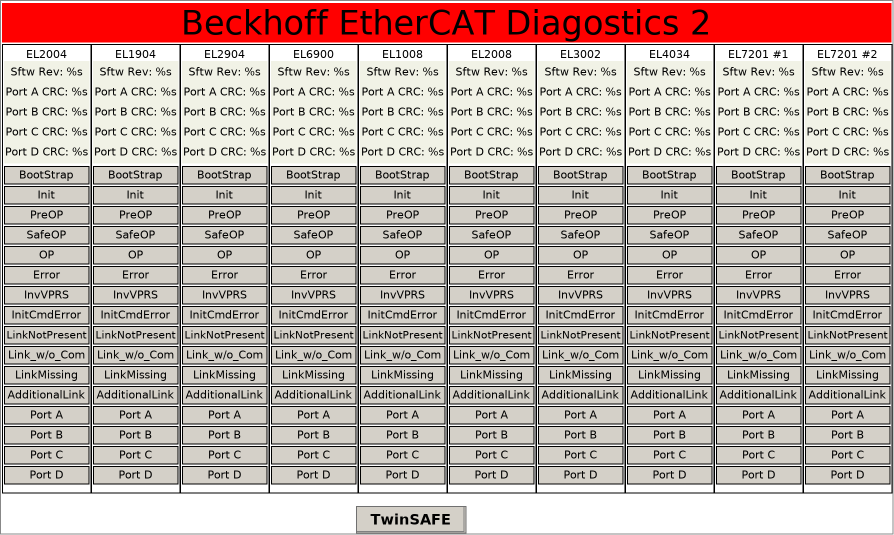
VISUALIZATION EtherCAT_Diag2  // 894x535
    Button (356,506 110x27), "TwinSAFE"
        OnMouseClick: change screen: TwinSAFE
    RoundedRectangle (2,3 889x39), "Beckhoff EtherCAT Diagostics 2"
    Group (2,42 89x451)
        RoundedRectangle (0,2 89x449)
        Label (2,0 85x25), "EL2004"
        Rectangle (2,19 85x22), "Sftw Rev: %s", text variable: g_iHMI_ProdCodeEL2004
        Rectangle (2,39 85x22), "Port A CRC: %s", text variable: g_stHMI_EL2004CrcErrorEx.portA
        Rectangle (2,59 85x22), "Port B CRC: %s", text variable: g_stHMI_EL2004CrcErrorEx.portB
        Rectangle (2,79 85x22), "Port C CRC: %s", text variable: g_stHMI_EL2004CrcErrorEx.portC
        Rectangle (2,99 85x22), "Port D CRC: %s", text variable: g_stHMI_EL2004CrcErrorEx.portD
        Rectangle (2,124 85x18), "BootStrap", colour toggle: g_stHMI_EL2004EcSlaveStateBits.bBootStrap
        Rectangle (2,144 85x18), "Init", colour toggle: g_stHMI_EL2004EcSlaveStateBits.bInit
        Rectangle (2,164 85x18), "PreOP", colour toggle: g_stHMI_EL2004EcSlaveStateBits.bPreop
        Rectangle (2,184 85x18), "SafeOP", colour toggle: g_stHMI_EL2004EcSlaveStateBits.bSafeOp
        Rectangle (2,204 85x18), "OP", colour toggle: g_stHMI_EL2004EcSlaveStateBits.bOp
        Rectangle (2,224 85x18), "Error", colour toggle: g_stHMI_EL2004EcSlaveStateBits.bError
        Rectangle (2,244 85x18), "InvVPRS", colour toggle: g_stHMI_EL2004EcSlaveStateBits.bInvVPRS
        Rectangle (2,264 85x18), "InitCmdError", colour toggle: g_stHMI_EL2004EcSlaveStateBits.bInitCmdError
        Rectangle (2,284 85x18), "LinkNotPresent", colour toggle: g_stHMI_EL2004EcSlaveStateBits.bLinkNotPresent
        Rectangle (2,304 85x18), "Link_w/o_Com", colour toggle: g_stHMI_EL2004EcSlaveStateBits.bLinkWithoutComm
        Rectangle (2,324 85x18), "LinkMissing", colour toggle: g_stHMI_EL2004EcSlaveStateBits.bLinkMissing
        Rectangle (2,344 85x18), "AdditionalLink", colour toggle: g_stHMI_EL2004EcSlaveStateBits.bAdditionalLink
        Rectangle (2,364 85x18), "Port A", colour toggle: g_stHMI_EL2004EcSlaveStateBits.bPortA
        Rectangle (2,384 85x18), "Port B", colour toggle: g_stHMI_EL2004EcSlaveStateBits.bPortB
        Rectangle (2,404 85x18), "Port C", colour toggle: g_stHMI_EL2004EcSlaveStateBits.bPortC
        Rectangle (2,424 85x18), "Port D", colour toggle: g_stHMI_EL2004EcSlaveStateBits.bPortD
    Group (91,42 89x451)
        RoundedRectangle (0,2 89x449)
        Label (2,0 85x25), "EL1904"
        Rectangle (2,19 85x22), "Sftw Rev: %s", text variable: g_iHMI_ProdCodeEL1904
        Rectangle (2,39 85x22), "Port A CRC: %s", text variable: g_stHMI_EL1904CrcErrorEx.portA
        Rectangle (2,59 85x22), "Port B CRC: %s", text variable: g_stHMI_EL1904CrcErrorEx.portB
        Rectangle (2,79 85x22), "Port C CRC: %s", text variable: g_stHMI_EL1904CrcErrorEx.portC
        Rectangle (2,99 85x22), "Port D CRC: %s", text variable: g_stHMI_EL1904CrcErrorEx.portD
        Rectangle (2,124 85x18), "BootStrap", colour toggle: g_stHMI_EL1904EcSlaveStateBits.bBootStrap
        Rectangle (2,144 85x18), "Init", colour toggle: g_stHMI_EL1904EcSlaveStateBits.bInit
        Rectangle (2,164 85x18), "PreOP", colour toggle: g_stHMI_EL1904EcSlaveStateBits.bPreop
        Rectangle (2,184 85x18), "SafeOP", colour toggle: g_stHMI_EL1904EcSlaveStateBits.bSafeOp
        Rectangle (2,204 85x18), "OP", colour toggle: g_stHMI_EL1904EcSlaveStateBits.bOp
        Rectangle (2,224 85x18), "Error", colour toggle: g_stHMI_EL1904EcSlaveStateBits.bError
        Rectangle (2,244 85x18), "InvVPRS", colour toggle: g_stHMI_EL1904EcSlaveStateBits.bInvVPRS
        Rectangle (2,264 85x18), "InitCmdError", colour toggle: g_stHMI_EL1904EcSlaveStateBits.bInitCmdError
        Rectangle (2,284 85x18), "LinkNotPresent", colour toggle: g_stHMI_EL1904EcSlaveStateBits.bLinkNotPresent
        Rectangle (2,304 85x18), "Link_w/o_Com", colour toggle: g_stHMI_EL1904EcSlaveStateBits.bLinkWithoutComm
        Rectangle (2,324 85x18), "LinkMissing", colour toggle: g_stHMI_EL1904EcSlaveStateBits.bLinkMissing
        Rectangle (2,344 85x18), "AdditionalLink", colour toggle: g_stHMI_EL1904EcSlaveStateBits.bAdditionalLink
        Rectangle (2,364 85x18), "Port A", colour toggle: g_stHMI_EL1904EcSlaveStateBits.bPortA
        Rectangle (2,384 85x18), "Port B", colour toggle: g_stHMI_EL1904EcSlaveStateBits.bPortB
        Rectangle (2,404 85x18), "Port C", colour toggle: g_stHMI_EL1904EcSlaveStateBits.bPortC
        Rectangle (2,424 85x18), "Port D", colour toggle: g_stHMI_EL1904EcSlaveStateBits.bPortD
    Group (180,42 89x451)
        RoundedRectangle (0,2 89x449)
        Label (2,0 85x25), "EL2904"
        Rectangle (2,19 85x22), "Sftw Rev: %s", text variable: g_iHMI_ProdCodeEL2904
        Rectangle (2,39 85x22), "Port A CRC: %s", text variable: g_stHMI_EL2904CrcErrorEx.portA
        Rectangle (2,59 85x22), "Port B CRC: %s", text variable: g_stHMI_EL2904CrcErrorEx.portB
        Rectangle (2,79 85x22), "Port C CRC: %s", text variable: g_stHMI_EL2904CrcErrorEx.portC
        Rectangle (2,99 85x22), "Port D CRC: %s", text variable: g_stHMI_EL2904CrcErrorEx.portD
        Rectangle (2,124 85x18), "BootStrap", colour toggle: g_stHMI_EL2904EcSlaveStateBits.bBootStrap
        Rectangle (2,144 85x18), "Init", colour toggle: g_stHMI_EL2904EcSlaveStateBits.bInit
        Rectangle (2,164 85x18), "PreOP", colour toggle: g_stHMI_EL2904EcSlaveStateBits.bPreop
        Rectangle (2,184 85x18), "SafeOP", colour toggle: g_stHMI_EL2904EcSlaveStateBits.bSafeOp
        Rectangle (2,204 85x18), "OP", colour toggle: g_stHMI_EL2904EcSlaveStateBits.bOp
        Rectangle (2,224 85x18), "Error", colour toggle: g_stHMI_EL2904EcSlaveStateBits.bError
        Rectangle (2,244 85x18), "InvVPRS", colour toggle: g_stHMI_EL2904EcSlaveStateBits.bInvVPRS
        Rectangle (2,264 85x18), "InitCmdError", colour toggle: g_stHMI_EL2904EcSlaveStateBits.bInitCmdError
        Rectangle (2,284 85x18), "LinkNotPresent", colour toggle: g_stHMI_EL2904EcSlaveStateBits.bLinkNotPresent
        Rectangle (2,304 85x18), "Link_w/o_Com", colour toggle: g_stHMI_EL2904EcSlaveStateBits.bLinkWithoutComm
        Rectangle (2,324 85x18), "LinkMissing", colour toggle: g_stHMI_EL2904EcSlaveStateBits.bLinkMissing
        Rectangle (2,344 85x18), "AdditionalLink", colour toggle: g_stHMI_EL2904EcSlaveStateBits.bAdditionalLink
        Rectangle (2,364 85x18), "Port A", colour toggle: g_stHMI_EL2904EcSlaveStateBits.bPortA
        Rectangle (2,384 85x18), "Port B", colour toggle: g_stHMI_EL2904EcSlaveStateBits.bPortB
        Rectangle (2,404 85x18), "Port C", colour toggle: g_stHMI_EL2904EcSlaveStateBits.bPortC
        Rectangle (2,424 85x18), "Port D", colour toggle: g_stHMI_EL2904EcSlaveStateBits.bPortD
    Group (269,42 89x451)
        RoundedRectangle (0,2 89x449)
        Label (2,0 85x25), "EL6900"
        Rectangle (2,19 85x22), "Sftw Rev: %s", text variable: g_iHMI_ProdCodeEL6900
        Rectangle (2,39 85x22), "Port A CRC: %s", text variable: g_stHMI_EL6900CrcErrorEx.portA
        Rectangle (2,59 85x22), "Port B CRC: %s", text variable: g_stHMI_EL6900CrcErrorEx.portB
        Rectangle (2,79 85x22), "Port C CRC: %s", text variable: g_stHMI_EL6900CrcErrorEx.portC
        Rectangle (2,99 85x22), "Port D CRC: %s", text variable: g_stHMI_EL6900CrcErrorEx.portD
        Rectangle (2,124 85x18), "BootStrap", colour toggle: g_stHMI_EL6900EcSlaveStateBits.bBootStrap
        Rectangle (2,144 85x18), "Init", colour toggle: g_stHMI_EL6900EcSlaveStateBits.bInit
        Rectangle (2,164 85x18), "PreOP", colour toggle: g_stHMI_EL6900EcSlaveStateBits.bPreop
        Rectangle (2,184 85x18), "SafeOP", colour toggle: g_stHMI_EL6900EcSlaveStateBits.bSafeOp
        Rectangle (2,204 85x18), "OP", colour toggle: g_stHMI_EL6900EcSlaveStateBits.bOp
        Rectangle (2,224 85x18), "Error", colour toggle: g_stHMI_EL6900EcSlaveStateBits.bError
        Rectangle (2,244 85x18), "InvVPRS", colour toggle: g_stHMI_EL6900EcSlaveStateBits.bInvVPRS
        Rectangle (2,264 85x18), "InitCmdError", colour toggle: g_stHMI_EL6900EcSlaveStateBits.bInitCmdError
        Rectangle (2,284 85x18), "LinkNotPresent", colour toggle: g_stHMI_EL6900EcSlaveStateBits.bLinkNotPresent
        Rectangle (2,304 85x18), "Link_w/o_Com", colour toggle: g_stHMI_EL6900EcSlaveStateBits.bLinkWithoutComm
        Rectangle (2,324 85x18), "LinkMissing", colour toggle: g_stHMI_EL6900EcSlaveStateBits.bLinkMissing
        Rectangle (2,344 85x18), "AdditionalLink", colour toggle: g_stHMI_EL6900EcSlaveStateBits.bAdditionalLink
        Rectangle (2,364 85x18), "Port A", colour toggle: g_stHMI_EL6900EcSlaveStateBits.bPortA
        Rectangle (2,384 85x18), "Port B", colour toggle: g_stHMI_EL6900EcSlaveStateBits.bPortB
        Rectangle (2,404 85x18), "Port C", colour toggle: g_stHMI_EL6900EcSlaveStateBits.bPortC
        Rectangle (2,424 85x18), "Port D", colour toggle: g_stHMI_EL6900EcSlaveStateBits.bPortD
    Group (358,42 89x451)
        RoundedRectangle (0,2 89x449)
        Label (2,0 85x25), "EL1008"
        Rectangle (2,19 85x22), "Sftw Rev: %s", text variable: g_iHMI_ProdCodeEL1008
        Rectangle (2,39 85x22), "Port A CRC: %s", text variable: g_stHMI_EL1008CrcErrorEx.portA
        Rectangle (2,59 85x22), "Port B CRC: %s", text variable: g_stHMI_EL1008CrcErrorEx.portB
        Rectangle (2,79 85x22), "Port C CRC: %s", text variable: g_stHMI_EL1008CrcErrorEx.portC
        Rectangle (2,99 85x22), "Port D CRC: %s", text variable: g_stHMI_EL1008CrcErrorEx.portD
        Rectangle (2,124 85x18), "BootStrap", colour toggle: g_stHMI_EL1008EcSlaveStateBits.bBootStrap
        Rectangle (2,144 85x18), "Init", colour toggle: g_stHMI_EL1008EcSlaveStateBits.bInit
        Rectangle (2,164 85x18), "PreOP", colour toggle: g_stHMI_EL1008EcSlaveStateBits.bPreop
        Rectangle (2,184 85x18), "SafeOP", colour toggle: g_stHMI_EL1008EcSlaveStateBits.bSafeOp
        Rectangle (2,204 85x18), "OP", colour toggle: g_stHMI_EL1008EcSlaveStateBits.bOp
        Rectangle (2,224 85x18), "Error", colour toggle: g_stHMI_EL1008EcSlaveStateBits.bError
        Rectangle (2,244 85x18), "InvVPRS", colour toggle: g_stHMI_EL1008EcSlaveStateBits.bInvVPRS
        Rectangle (2,264 85x18), "InitCmdError", colour toggle: g_stHMI_EL1008EcSlaveStateBits.bInitCmdError
        Rectangle (2,284 85x18), "LinkNotPresent", colour toggle: g_stHMI_EL1008EcSlaveStateBits.bLinkNotPresent
        Rectangle (2,304 85x18), "Link_w/o_Com", colour toggle: g_stHMI_EL1008EcSlaveStateBits.bLinkWithoutComm
        Rectangle (2,324 85x18), "LinkMissing", colour toggle: g_stHMI_EL1008EcSlaveStateBits.bLinkMissing
        Rectangle (2,344 85x18), "AdditionalLink", colour toggle: g_stHMI_EL1008EcSlaveStateBits.bAdditionalLink
        Rectangle (2,364 85x18), "Port A", colour toggle: g_stHMI_EL1008EcSlaveStateBits.bPortA
        Rectangle (2,384 85x18), "Port B", colour toggle: g_stHMI_EL1008EcSlaveStateBits.bPortB
        Rectangle (2,404 85x18), "Port C", colour toggle: g_stHMI_EL1008EcSlaveStateBits.bPortC
        Rectangle (2,424 85x18), "Port D", colour toggle: g_stHMI_EL1008EcSlaveStateBits.bPortD
    Group (447,42 89x451)
        RoundedRectangle (0,2 89x449)
        Label (2,0 85x25), "EL2008"
        Rectangle (2,19 85x22), "Sftw Rev: %s", text variable: g_iHMI_ProdCodeEL2008
        Rectangle (2,39 85x22), "Port A CRC: %s", text variable: g_stHMI_EL2008CrcErrorEx.portA
        Rectangle (2,59 85x22), "Port B CRC: %s", text variable: g_stHMI_EL2008CrcErrorEx.portB
        Rectangle (2,79 85x22), "Port C CRC: %s", text variable: g_stHMI_EL2008CrcErrorEx.portC
        Rectangle (2,99 85x22), "Port D CRC: %s", text variable: g_stHMI_EL2008CrcErrorEx.portD
        Rectangle (2,124 85x18), "BootStrap", colour toggle: g_stHMI_EL2008EcSlaveStateBits.bBootStrap
        Rectangle (2,144 85x18), "Init", colour toggle: g_stHMI_EL2008EcSlaveStateBits.bInit
        Rectangle (2,164 85x18), "PreOP", colour toggle: g_stHMI_EL2008EcSlaveStateBits.bPreop
        Rectangle (2,184 85x18), "SafeOP", colour toggle: g_stHMI_EL2008EcSlaveStateBits.bSafeOp
        Rectangle (2,204 85x18), "OP", colour toggle: g_stHMI_EL2008EcSlaveStateBits.bOp
        Rectangle (2,224 85x18), "Error", colour toggle: g_stHMI_EL2008EcSlaveStateBits.bError
        Rectangle (2,244 85x18), "InvVPRS", colour toggle: g_stHMI_EL2008EcSlaveStateBits.bInvVPRS
        Rectangle (2,264 85x18), "InitCmdError", colour toggle: g_stHMI_EL2008EcSlaveStateBits.bInitCmdError
        Rectangle (2,284 85x18), "LinkNotPresent", colour toggle: g_stHMI_EL2008EcSlaveStateBits.bLinkNotPresent
        Rectangle (2,304 85x18), "Link_w/o_Com", colour toggle: g_stHMI_EL2008EcSlaveStateBits.bLinkWithoutComm
        Rectangle (2,324 85x18), "LinkMissing", colour toggle: g_stHMI_EL2008EcSlaveStateBits.bLinkMissing
        Rectangle (2,344 85x18), "AdditionalLink", colour toggle: g_stHMI_EL2008EcSlaveStateBits.bAdditionalLink
        Rectangle (2,364 85x18), "Port A", colour toggle: g_stHMI_EL2008EcSlaveStateBits.bPortA
        Rectangle (2,384 85x18), "Port B", colour toggle: g_stHMI_EL2008EcSlaveStateBits.bPortB
        Rectangle (2,404 85x18), "Port C", colour toggle: g_stHMI_EL2008EcSlaveStateBits.bPortC
        Rectangle (2,424 85x18), "Port D", colour toggle: g_stHMI_EL2008EcSlaveStateBits.bPortD
    Group (536,42 89x451)
        RoundedRectangle (0,2 89x449)
        Label (2,0 85x25), "EL3002"
        Rectangle (2,19 85x22), "Sftw Rev: %s", text variable: g_iHMI_ProdCodeEL3002
        Rectangle (2,39 85x22), "Port A CRC: %s", text variable: g_stHMI_EL3002CrcErrorEx.portA
        Rectangle (2,59 85x22), "Port B CRC: %s", text variable: g_stHMI_EL3002CrcErrorEx.portB
        Rectangle (2,79 85x22), "Port C CRC: %s", text variable: g_stHMI_EL3002CrcErrorEx.portC
        Rectangle (2,99 85x22), "Port D CRC: %s", text variable: g_stHMI_EL3002CrcErrorEx.portD
        Rectangle (2,124 85x18), "BootStrap", colour toggle: g_stHMI_EL3002EcSlaveStateBits.bBootStrap
        Rectangle (2,144 85x18), "Init", colour toggle: g_stHMI_EL3002EcSlaveStateBits.bInit
        Rectangle (2,164 85x18), "PreOP", colour toggle: g_stHMI_EL3002EcSlaveStateBits.bPreop
        Rectangle (2,184 85x18), "SafeOP", colour toggle: g_stHMI_EL3002EcSlaveStateBits.bSafeOp
        Rectangle (2,204 85x18), "OP", colour toggle: g_stHMI_EL3002EcSlaveStateBits.bOp
        Rectangle (2,224 85x18), "Error", colour toggle: g_stHMI_EL3002EcSlaveStateBits.bError
        Rectangle (2,244 85x18), "InvVPRS", colour toggle: g_stHMI_EL3002EcSlaveStateBits.bInvVPRS
        Rectangle (2,264 85x18), "InitCmdError", colour toggle: g_stHMI_EL3002EcSlaveStateBits.bInitCmdError
        Rectangle (2,284 85x18), "LinkNotPresent", colour toggle: g_stHMI_EL3002EcSlaveStateBits.bLinkNotPresent
        Rectangle (2,304 85x18), "Link_w/o_Com", colour toggle: g_stHMI_EL3002EcSlaveStateBits.bLinkWithoutComm
        Rectangle (2,324 85x18), "LinkMissing", colour toggle: g_stHMI_EL3002EcSlaveStateBits.bLinkMissing
        Rectangle (2,344 85x18), "AdditionalLink", colour toggle: g_stHMI_EL3002EcSlaveStateBits.bAdditionalLink
        Rectangle (2,364 85x18), "Port A", colour toggle: g_stHMI_EL3002EcSlaveStateBits.bPortA
        Rectangle (2,384 85x18), "Port B", colour toggle: g_stHMI_EL3002EcSlaveStateBits.bPortB
        Rectangle (2,404 85x18), "Port C", colour toggle: g_stHMI_EL3002EcSlaveStateBits.bPortC
        Rectangle (2,424 85x18), "Port D", colour toggle: g_stHMI_EL3002EcSlaveStateBits.bPortD
    Group (625,42 89x451)
        RoundedRectangle (0,2 89x449)
        Label (2,0 85x25), "EL4034"
        Rectangle (2,19 85x22), "Sftw Rev: %s", text variable: g_iHMI_ProdCodeEL4034
        Rectangle (2,39 85x22), "Port A CRC: %s", text variable: g_stHMI_EL4034CrcErrorEx.portA
        Rectangle (2,59 85x22), "Port B CRC: %s", text variable: g_stHMI_EL4034CrcErrorEx.portB
        Rectangle (2,79 85x22), "Port C CRC: %s", text variable: g_stHMI_EL4034CrcErrorEx.portC
        Rectangle (2,99 85x22), "Port D CRC: %s", text variable: g_stHMI_EL4034CrcErrorEx.portD
        Rectangle (2,124 85x18), "BootStrap", colour toggle: g_stHMI_EL4034EcSlaveStateBits.bBootStrap
        Rectangle (2,144 85x18), "Init", colour toggle: g_stHMI_EL4034EcSlaveStateBits.bInit
        Rectangle (2,164 85x18), "PreOP", colour toggle: g_stHMI_EL4034EcSlaveStateBits.bPreop
        Rectangle (2,184 85x18), "SafeOP", colour toggle: g_stHMI_EL4034EcSlaveStateBits.bSafeOp
        Rectangle (2,204 85x18), "OP", colour toggle: g_stHMI_EL4034EcSlaveStateBits.bOp
        Rectangle (2,224 85x18), "Error", colour toggle: g_stHMI_EL4034EcSlaveStateBits.bError
        Rectangle (2,244 85x18), "InvVPRS", colour toggle: g_stHMI_EL4034EcSlaveStateBits.bInvVPRS
        Rectangle (2,264 85x18), "InitCmdError", colour toggle: g_stHMI_EL4034EcSlaveStateBits.bInitCmdError
        Rectangle (2,284 85x18), "LinkNotPresent", colour toggle: g_stHMI_EL4034EcSlaveStateBits.bLinkNotPresent
        Rectangle (2,304 85x18), "Link_w/o_Com", colour toggle: g_stHMI_EL4034EcSlaveStateBits.bLinkWithoutComm
        Rectangle (2,324 85x18), "LinkMissing", colour toggle: g_stHMI_EL4034EcSlaveStateBits.bLinkMissing
        Rectangle (2,344 85x18), "AdditionalLink", colour toggle: g_stHMI_EL4034EcSlaveStateBits.bAdditionalLink
        Rectangle (2,364 85x18), "Port A", colour toggle: g_stHMI_EL4034EcSlaveStateBits.bPortA
        Rectangle (2,384 85x18), "Port B", colour toggle: g_stHMI_EL4034EcSlaveStateBits.bPortB
        Rectangle (2,404 85x18), "Port C", colour toggle: g_stHMI_EL4034EcSlaveStateBits.bPortC
        Rectangle (2,424 85x18), "Port D", colour toggle: g_stHMI_EL4034EcSlaveStateBits.bPortD
    Group (714,42 89x451)
        RoundedRectangle (0,2 89x449)
        Label (2,0 85x25), "EL7201 #1"
        Rectangle (2,19 85x22), "Sftw Rev: %s", text variable: g_iHMI_ProdCodeEL7201_1
        Rectangle (2,39 85x22), "Port A CRC: %s", text variable: g_stHMI_EL7201_1CrcErrorEx.portA
        Rectangle (2,59 85x22), "Port B CRC: %s", text variable: g_stHMI_EL7201_1CrcErrorEx.portB
        Rectangle (2,79 85x22), "Port C CRC: %s", text variable: g_stHMI_EL7201_1CrcErrorEx.portC
        Rectangle (2,99 85x22), "Port D CRC: %s", text variable: g_stHMI_EL7201_1CrcErrorEx.portD
        Rectangle (2,124 85x18), "BootStrap", colour toggle: g_stHMI_EL7201_1EcSlaveStateBits.bBootStrap
        Rectangle (2,144 85x18), "Init", colour toggle: g_stHMI_EL7201_1EcSlaveStateBits.bInit
        Rectangle (2,164 85x18), "PreOP", colour toggle: g_stHMI_EL7201_1EcSlaveStateBits.bPreop
        Rectangle (2,184 85x18), "SafeOP", colour toggle: g_stHMI_EL7201_1EcSlaveStateBits.bSafeOp
        Rectangle (2,204 85x18), "OP", colour toggle: g_stHMI_EL7201_1EcSlaveStateBits.bOp
        Rectangle (2,224 85x18), "Error", colour toggle: g_stHMI_EL7201_1EcSlaveStateBits.bError
        Rectangle (2,244 85x18), "InvVPRS", colour toggle: g_stHMI_EL7201_1EcSlaveStateBits.bInvVPRS
        Rectangle (2,264 85x18), "InitCmdError", colour toggle: g_stHMI_EL7201_1EcSlaveStateBits.bInitCmdError
        Rectangle (2,284 85x18), "LinkNotPresent", colour toggle: g_stHMI_EL7201_1EcSlaveStateBits.bLinkNotPresent
        Rectangle (2,304 85x18), "Link_w/o_Com", colour toggle: g_stHMI_EL7201_1EcSlaveStateBits.bLinkWithoutComm
        Rectangle (2,324 85x18), "LinkMissing", colour toggle: g_stHMI_EL7201_1EcSlaveStateBits.bLinkMissing
        Rectangle (2,344 85x18), "AdditionalLink", colour toggle: g_stHMI_EL7201_1EcSlaveStateBits.bAdditionalLink
        Rectangle (2,364 85x18), "Port A", colour toggle: g_stHMI_EL7201_1EcSlaveStateBits.bPortA
        Rectangle (2,384 85x18), "Port B", colour toggle: g_stHMI_EL7201_1EcSlaveStateBits.bPortB
        Rectangle (2,404 85x18), "Port C", colour toggle: g_stHMI_EL7201_1EcSlaveStateBits.bPortC
        Rectangle (2,424 85x18), "Port D", colour toggle: g_stHMI_EL7201_1EcSlaveStateBits.bPortD
    Group (803,42 89x451)
        RoundedRectangle (0,2 89x449)
        Label (2,0 85x25), "EL7201 #2"
        Rectangle (2,19 85x22), "Sftw Rev: %s", text variable: g_iHMI_ProdCodeEL7201_2
        Rectangle (2,39 85x22), "Port A CRC: %s", text variable: g_stHMI_EL7201_2CrcErrorEx.portA
        Rectangle (2,59 85x22), "Port B CRC: %s", text variable: g_stHMI_EL7201_2CrcErrorEx.portB
        Rectangle (2,79 85x22), "Port C CRC: %s", text variable: g_stHMI_EL7201_2CrcErrorEx.portC
        Rectangle (2,99 85x22), "Port D CRC: %s", text variable: g_stHMI_EL7201_2CrcErrorEx.portD
        Rectangle (2,124 85x18), "BootStrap", colour toggle: g_stHMI_EL7201_2EcSlaveStateBits.bBootStrap
        Rectangle (2,144 85x18), "Init", colour toggle: g_stHMI_EL7201_2EcSlaveStateBits.bInit
        Rectangle (2,164 85x18), "PreOP", colour toggle: g_stHMI_EL7201_2EcSlaveStateBits.bPreop
        Rectangle (2,184 85x18), "SafeOP", colour toggle: g_stHMI_EL7201_2EcSlaveStateBits.bSafeOp
        Rectangle (2,204 85x18), "OP", colour toggle: g_stHMI_EL7201_2EcSlaveStateBits.bOp
        Rectangle (2,224 85x18), "Error", colour toggle: g_stHMI_EL7201_2EcSlaveStateBits.bError
        Rectangle (2,244 85x18), "InvVPRS", colour toggle: g_stHMI_EL7201_2EcSlaveStateBits.bInvVPRS
        Rectangle (2,264 85x18), "InitCmdError", colour toggle: g_stHMI_EL7201_2EcSlaveStateBits.bInitCmdError
        Rectangle (2,284 85x18), "LinkNotPresent", colour toggle: g_stHMI_EL7201_2EcSlaveStateBits.bLinkNotPresent
        Rectangle (2,304 85x18), "Link_w/o_Com", colour toggle: g_stHMI_EL7201_2EcSlaveStateBits.bLinkWithoutComm
        Rectangle (2,324 85x18), "LinkMissing", colour toggle: g_stHMI_EL7201_2EcSlaveStateBits.bLinkMissing
        Rectangle (2,344 85x18), "AdditionalLink", colour toggle: g_stHMI_EL7201_2EcSlaveStateBits.bAdditionalLink
        Rectangle (2,364 85x18), "Port A", colour toggle: g_stHMI_EL7201_2EcSlaveStateBits.bPortA
        Rectangle (2,384 85x18), "Port B", colour toggle: g_stHMI_EL7201_2EcSlaveStateBits.bPortB
        Rectangle (2,404 85x18), "Port C", colour toggle: g_stHMI_EL7201_2EcSlaveStateBits.bPortC
        Rectangle (2,424 85x18), "Port D", colour toggle: g_stHMI_EL7201_2EcSlaveStateBits.bPortD
END_VISUALIZATION

(* stored: Version 1.1.0.1, ProductVersion 3.1.0.18
   Visu EtherCAT_Diag2: Id {c47ef602-3c17-4ba1-af93-d5a8736ac622} *)
